# EPICS substitutions: iocBoot/iocDera/motor.substitutions
file "$(MOTOR)/db/asyn_motor.db"
{
pattern
{P,    N,   M,         DTYP,      PORT,   ADDR, DESC, EGU,  DIR,  VELO,  VBAS, ACCL, BDST, BVEL, BACC,    MRES,       PREC, DHLM, DLLM, INIT}
# Newport NSA12 stage, 6.35 microns/full step, 128 micro-steps/s
{Dera:, 1, "m$(N)", "asynMotor",  CONEX1,    0, "X",    mm,  Pos,   1.,    0.1,  .25,    0,    1,   .2,  4.9609375e-5,   4,   11,   0,   ""}
{Dera:, 2, "m$(N)", "asynMotor",  CONEX2,    0, "Y",    mm,  Pos,   1.,    0.1,  .25,    0,    1,   .2,  4.9609375e-5,   4,   11,   0,   ""}
{Dera:, 3, "m$(N)", "asynMotor",  CONEX3,    0, "Z",    mm,  Pos,   1.,    0.1,  .25,    0,    1,   .2,  4.9609375e-5,   4,   11,   0,   ""}
}
